Fanuc KAREL source: IO0088.KL

-- PROVISIONAL review KL for V1013-1; original PC SHA256 dbebcd24c2c3861dc105848ca1d6dda9050dcfa10dbaca746abc8e6102e35192
-- Incomplete behavior may be omitted. Consult companion uncertainty JSON. Do not deploy.
PROGRAM IO0088
%NOLOCKGROUP
-- UNRESOLVED_LOCAL_POOL 5 cells at code offset 13; source declarations unknown
-- DIRECT_LOCAL_WORD_ACCESS alone does not prove INTEGER, REAL, or BOOLEAN
BEGIN
  -- UNRESOLVED_PC offsets 0-18; opcodes 2B,2C,7B
  -- UNRESOLVED_PC offsets 23-30; opcodes 9D,23
  -- UNRESOLVED_PC offsets 35-49; opcodes 2E,22,9D,33,35
  -- UNRESOLVED_PC offsets 54-61; opcodes 9D,23
  -- UNRESOLVED_PC offsets 66-77; opcodes 2E,23
  -- UNRESOLVED_PC offsets 82-99; opcodes 21,9D,52,19,64,23
  -- UNRESOLVED_PC offsets 104-108; opcodes 7F
  -- UNRESOLVED_PC offsets 113-117; opcodes 27,AA
  -- UNRESOLVED_PC offsets 122-126; opcodes 7F
END IO0088
